Fanuc KAREL source: SIN.kl

PROGRAM T
%NOLOCKGROUP
VAR
 v0 : REAL
 res : REAL
BEGIN
 res = SIN(v0)
END T
